FUNCTION_BLOCK Station_CAT (* Composite Function Block Type *)
  (* Standard: 61499-2 *)
  (* Version 0.0, 7/31/2025, Evans_A, Schneider Electric, template *)
  PACKAGE Main;
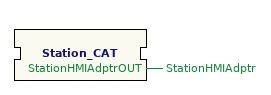
  PLUGS
    StationHMIAdptrOUT : StationHMIAdptr;
  END_PLUGS
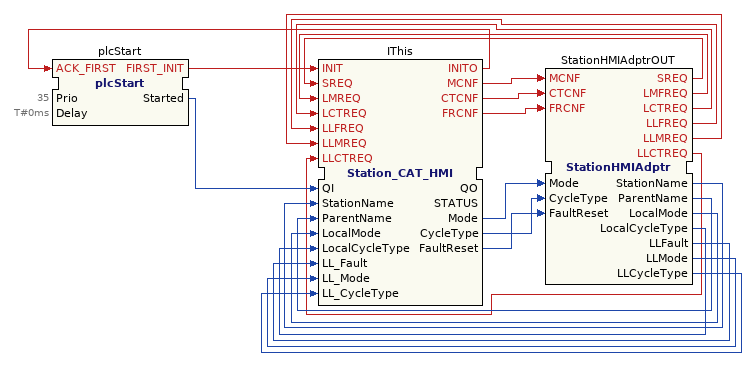
  FBS
    IThis : Station_CAT_HMI;
    plcStart : plcStart(Prio := 35, Delay := T#0ms);
  END_FBS
  EVENT_CONNECTIONS
    plcStart.FIRST_INIT TO IThis.INIT;
    IThis.INITO TO plcStart.ACK_FIRST;
    IThis.MCNF TO StationHMIAdptrOUT.MCNF;
    IThis.CTCNF TO StationHMIAdptrOUT.CTCNF;
    IThis.FRCNF TO StationHMIAdptrOUT.FRCNF;
    StationHMIAdptrOUT.SREQ TO IThis.SREQ;
    StationHMIAdptrOUT.LMFREQ TO IThis.LMREQ;
    StationHMIAdptrOUT.LCTREQ TO IThis.LCTREQ;
    StationHMIAdptrOUT.LLFREQ TO IThis.LLFREQ;
    StationHMIAdptrOUT.LLMREQ TO IThis.LLMREQ;
    StationHMIAdptrOUT.LLCTREQ TO IThis.LLCTREQ;
  END_CONNECTIONS
  DATA_CONNECTIONS
    plcStart.Started TO IThis.QI;
    IThis.Mode TO StationHMIAdptrOUT.Mode;
    IThis.CycleType TO StationHMIAdptrOUT.CycleType;
    IThis.FaultReset TO StationHMIAdptrOUT.FaultReset;
    StationHMIAdptrOUT.StationName TO IThis.StationName;
    StationHMIAdptrOUT.ParentName TO IThis.ParentName;
    StationHMIAdptrOUT.LocalMode TO IThis.LocalMode;
    StationHMIAdptrOUT.LocalCycleType TO IThis.LocalCycleType;
    StationHMIAdptrOUT.LLFault TO IThis.LL_Fault;
    StationHMIAdptrOUT.LLMode TO IThis.LL_Mode;
    StationHMIAdptrOUT.LLCycleType TO IThis.LL_CycleType;
  END_CONNECTIONS
END_FUNCTION_BLOCK
